// TIA Portal V15.1 export
// export: Created 2020-06-12T07:35:43.3505859Z, ExportSetting None, DisplayName Totally Integrated Automation Portal, DisplayVersion V15.1, DisplayName TIA Portal Openness, DisplayVersion V15.1, DisplayName STEP 7 Professional, DisplayVersion V15.1, DisplayName STEP 7 Safety, DisplayVersion V15.1, DisplayName WinCC Advanced, DisplayVersion V15.1
FUNCTION "CW_Tank" : Void   // FC117, FBD
{ S7_Optimized_Access := 'TRUE' }
// stored: SetENOAutomatically False
   VAR_TEMP
      tPRS_to_m : Real;
      tHeat_rel : Bool;
      tCV01set : Real;
      _temp_off : Real;
      _temp_on : Real;
      tReqTankFillStart : Bool;
      tReqTankFillStop : Bool;
      tWaterLevel : Real;
      tCVMin : Real;
      tCVMax : Real;
   END_VAR
   VAR_TEMP   // added for the SCL form of the ladder/FBD networks
      _w1 : Bool;
   END_VAR
BEGIN

REGION Network 1: HMI request treat
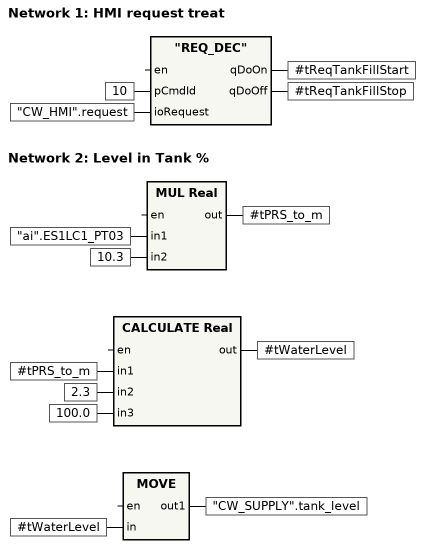
   "REQ_DEC"(pCmdId := 10,
             ioRequest := "CW_HMI".request,
             qDoOn => #tReqTankFillStart,
             qDoOff => #tReqTankFillStop);
END_REGION

REGION Network 2: Level in Tank %
   #tPRS_to_m := "ai".ES1LC1_PT03 * 10.3;
   #tWaterLevel := #tPRS_to_m/2.3*100.0;
   "CW_SUPPLY".tank_level := #tWaterLevel;
END_REGION

REGION Network 3: Detects defined levels of water in the tank
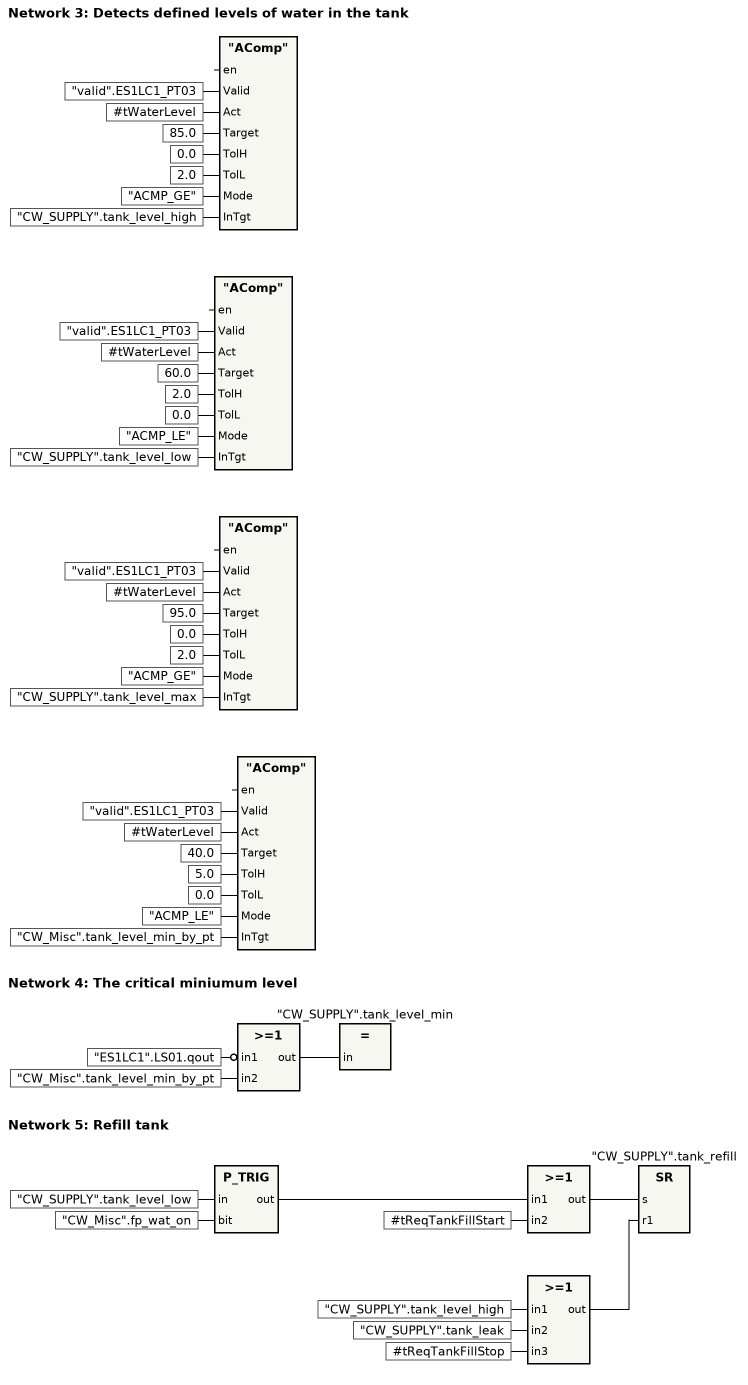
   "AComp"(Valid := "valid".ES1LC1_PT03,
           Act := #tWaterLevel,
           Target := 85.0,
           TolH := 0.0,
           TolL := 2.0,
           Mode := "ACMP_GE",
           InTgt := "CW_SUPPLY".tank_level_high);
   "AComp"(Valid := "valid".ES1LC1_PT03,
           Act := #tWaterLevel,
           Target := 60.0,
           TolH := 2.0,
           TolL := 0.0,
           Mode := "ACMP_LE",
           InTgt := "CW_SUPPLY".tank_level_low);
   "AComp"(Valid := "valid".ES1LC1_PT03,
           Act := #tWaterLevel,
           Target := 95.0,
           TolH := 0.0,
           TolL := 2.0,
           Mode := "ACMP_GE",
           InTgt := "CW_SUPPLY".tank_level_max);
   "AComp"(Valid := "valid".ES1LC1_PT03,
           Act := #tWaterLevel,
           Target := 40.0,
           TolH := 5.0,
           TolL := 0.0,
           Mode := "ACMP_LE",
           InTgt := "CW_Misc".tank_level_min_by_pt);
END_REGION

REGION Network 4: The critical miniumum level
   "CW_SUPPLY".tank_level_min := NOT "ES1LC1".LS01.qout OR "CW_Misc".tank_level_min_by_pt;
END_REGION

REGION Network 5: Refill tank
   // start =1.8
   // stop =2.0
   #_w1 := "CW_SUPPLY".tank_level_low AND NOT "CW_Misc".fp_wat_on;   // rising edge
   "CW_Misc".fp_wat_on := "CW_SUPPLY".tank_level_low;
   IF #_w1 OR #tReqTankFillStart THEN
       "CW_SUPPLY".tank_refill := TRUE;   // SR flip-flop
   END_IF;
   IF "CW_SUPPLY".tank_level_high OR "CW_SUPPLY".tank_leak OR #tReqTankFillStop THEN
       "CW_SUPPLY".tank_refill := FALSE;
   END_IF;
END_REGION

REGION Network 6: Tank leakage detection during refilling
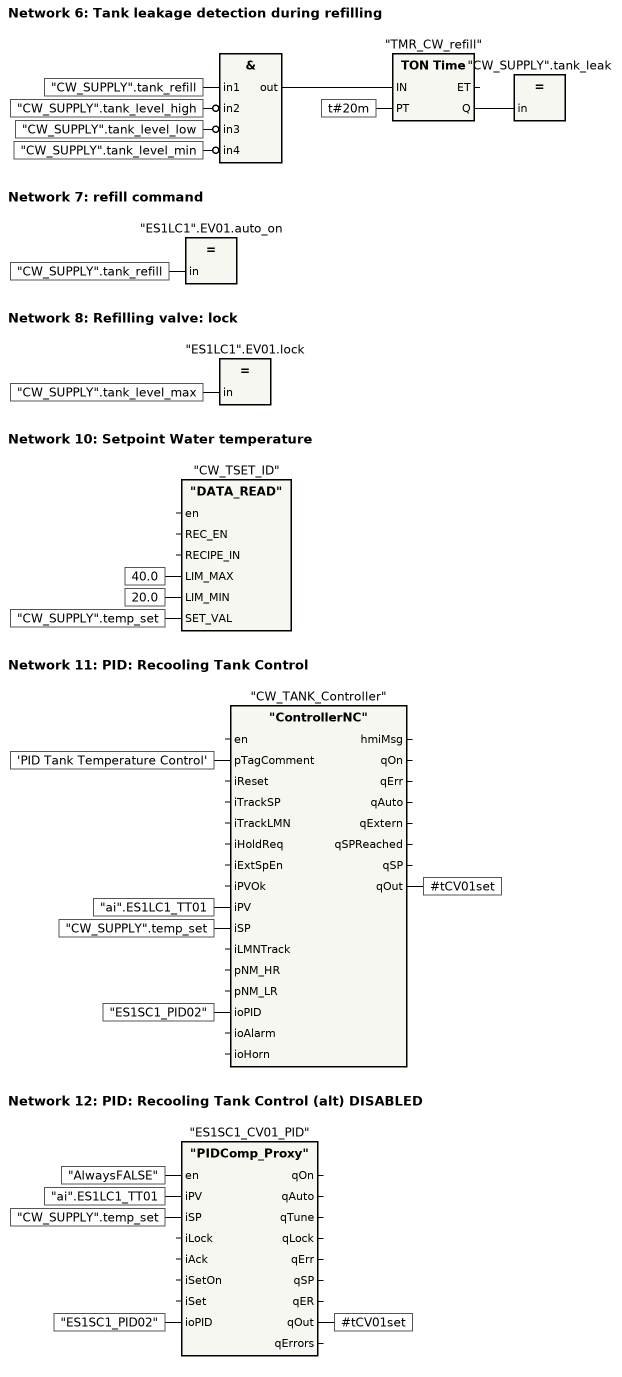
   "TMR_CW_refill".TON(IN := "CW_SUPPLY".tank_refill AND NOT "CW_SUPPLY".tank_level_high AND NOT "CW_SUPPLY".tank_level_low AND NOT "CW_SUPPLY".tank_level_min,
                       PT := t#20m);
   "CW_SUPPLY".tank_leak := "TMR_CW_refill".Q;
END_REGION

REGION Network 7: refill command
   "ES1LC1".EV01.auto_on := "CW_SUPPLY".tank_refill;
END_REGION

REGION Network 8: Refilling valve: lock
   "ES1LC1".EV01.lock := "CW_SUPPLY".tank_level_max;
END_REGION

REGION Network 9: ### Temperature control ###
END_REGION

REGION Network 10: Setpoint Water temperature
   "CW_TSET_ID"(LIM_MAX := 40.0, LIM_MIN := 20.0, SET_VAL := "CW_SUPPLY".temp_set);   // "DATA_READ"
END_REGION

REGION Network 11: PID: Recooling Tank Control
   "CW_TANK_Controller"(pTagComment := 'PID Tank Temperature Control',   // "ControllerNC"
                        iPV := "ai".ES1LC1_TT01,
                        iSP := "CW_SUPPLY".temp_set,
                        ioPID := "ES1SC1_PID02",
                        qOut => #tCV01set);
END_REGION

REGION Network 12: PID: Recooling Tank Control (alt) DISABLED
   IF "AlwaysFALSE" THEN
       "ES1SC1_CV01_PID"(iPV := "ai".ES1LC1_TT01,   // "PIDComp_Proxy"
                         iSP := "CW_SUPPLY".temp_set,
                         ioPID := "ES1SC1_PID02",
                         qOut => #tCV01set);
   END_IF;
END_REGION

REGION Network 13: To Output
   // That is not good idea to fully close CV
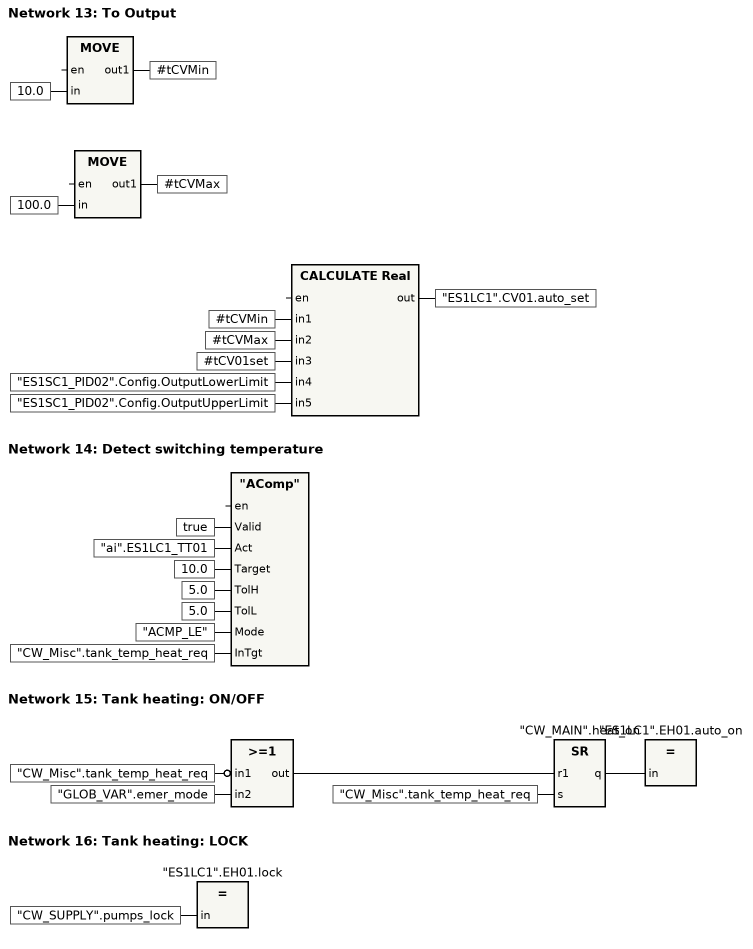
   #tCVMin := 10.0;
   #tCVMax := 100.0;
   "ES1LC1".CV01.auto_set := #tCVMax - (#tCVMin + (#tCVMax - #tCVMin) * ((#tCV01set - "ES1SC1_PID02".Config.OutputLowerLimit) / ("ES1SC1_PID02".Config.OutputUpperLimit - "ES1SC1_PID02".Config.OutputLowerLimit)));
END_REGION

REGION Network 14: Detect switching temperature
   "AComp"(Valid := true,
           Act := "ai".ES1LC1_TT01,
           Target := 10.0,
           TolH := 5.0,
           TolL := 5.0,
           Mode := "ACMP_LE",
           InTgt := "CW_Misc".tank_temp_heat_req);
END_REGION

REGION Network 15: Tank heating: ON/OFF
   IF "CW_Misc".tank_temp_heat_req THEN
       "CW_MAIN".heat_on := TRUE;   // SR flip-flop
   END_IF;
   IF NOT "CW_Misc".tank_temp_heat_req OR "GLOB_VAR".emer_mode THEN "CW_MAIN".heat_on := FALSE; END_IF;
   "ES1LC1".EH01.auto_on := "CW_MAIN".heat_on;
END_REGION

REGION Network 16: Tank heating: LOCK
   "ES1LC1".EH01.lock := "CW_SUPPLY".pumps_lock;
END_REGION
END_FUNCTION
